{attribute 'GeneratedUsingTerminal: EK1100-0000-0018'}
{attribute addProperty BoxType "EK1100-0000-0018"}
{attribute addProperty Id "Term_882_EL1809EL1809_32157CFD20Term_883_EL1809EL1809_32157CFD20Term_884_EL1809EL1809_32157CFD20Term_885_EL1809EL1809_32157CFD20Term_886_EL1809EL1809_32157CFD20Term_887_EL1809EL1809_32157CFD20Term_888_EL1809EL1809_32157CFD20Term_889_EL1809EL1809_32157CFD20Term_890_EL1809EL1809_32157CFD20Term_891_EL1809EL1809_32157CFD20Term_892_EL1809EL1809_32157CFD20Term_893_EL1809EL1809_32157CFD20Term_894_EL1809EL1809_32157CFD20Term_895_EL1809EL1809_32157CFD20Term_896_EL1809EL1809_32157CFD20Term_897_EL1809EL1809_32157CFD20Term_898_EL1809EL1809_32157CFD20Term_899_EL1809EL1809_32157CFD20Term_900_EL1809EL1809_32157CFD20Term_901_EL1809EL1809_32157CFD20Term_902_EL1809EL1809_32157CFD20Term_903_EL1809EL1809_32157CFD20Term_904_EL1809EL1809_32157CFD20Term_905_EL1809EL1809_32157CFD20Term_906_EL1809EL1809_32157CFD20Term_933_EL1809EL1809_32157CFD20Term_934_EL1809EL1809_32157CFD20Term_935_EL1809EL1809_32157CFD20Term_936_EL1809EL1809_32157CFD20Term_937_EL1809EL1809_32157CFD20Term_938_EL1809EL1809_32157CFD20Term_939_EL1809EL1809_32157CFD20Term_940_EL1809EL1809_32157CFD20Term_941_EL1809EL1809_32157CFD20Term_942_EL1809EL1809_32157CFD20Term_943_EL1809EL1809_32157CFD20Term_944_EL1809EL1809_32157CFD20Term_945_EL1809EL1809_32157CFD20Term_946_EL1809EL1809_32157CFD20Term_947_EL1809EL1809_32157CFD20Term_948_EL1809EL1809_32157CFD20Term_949_EL1809EL1809_32157CFD20Term_950_EL1809EL1809_32157CFD20Term_951_EL1809EL1809_32157CFD20Term_952_EL1809EL1809_32157CFD20Term_953_EL1809EL1809_32157CFD20Term_954_EL1809EL1809_32157CFD20Term_955_EL1809EL1809_32157CFD20Term_956_EL1809EL1809_32157CFD20Term_957_EL1809EL1809_32157CFD20Term_958_EL1809EL1809_32157CFD20Term_959_EL1809EL1809_32157CFD20Term_960_EL1809EL1809_32157CFD20Term_961_EL1809EL1809_32157CFD20Term_962_EL1809EL1809_32157CFD20Term_963_EL1809EL1809_32157CFD20Term_964_EL1809EL1809_32157CFD20Term_965_EL1809EL1809_32157CFD20Term_967_EL1809EL1809_32157CFD20Term_968_EL1809EL1809_32157CFD20Term_969_EL1809EL1809_32157CFD20Term_970_EL1809EL1809_32157CFD20Term_971_EL1809EL1809_32157CFD20Term_972_EL1809EL1809_32157CFD20Term_973_EL1809EL1809_32157CFD20Term_974_EL1809EL1809_32157CFD20Term_975_EL1809EL1809_32157CFD20Term_976_EL1809EL1809_32157CFD20Term_977_EL1809EL1809_32157CFD20Term_978_EL1809EL1809_32157CFD20Term_979_EL1809EL1809_32157CFD20Term_980_EL1809EL1809_32157CFD20Term_981_EL1809EL1809_32157CFD20Term_982_EL1809EL1809_32157CFD20Term_983_EL1809EL1809_32157CFD20Term_984_EL1809EL1809_32157CFD20Term_986_EL1809EL1809_32157CFD20Term_987_EL1809EL1809_32157CFD20Term_988_EL1809EL1809_32157CFD20Term_989_EL1809EL1809_32157CFD20Term_1025_EL1809EL1809_32157CFD20Term_1026_EL1809EL1809_32157CFD20Term_1027_EL1809EL1809_32157CFD20Term_1028_EL1809EL1809_32157CFD20Term_1029_EL1809EL1809_32157CFD20Term_1030_EL1809EL1809_32157CFD20Term_1031_EL1809EL1809_32157CFD20Term_1032_EL1809EL1809_32157CFD20Term_1033_EL1809EL1809_32157CFD20Term_1034_EL1809EL1809_32157CFD20Term_1035_EL1809EL1809_32157CFD20Term_1036_EL1809EL1809_32157CFD20Term_1038_EL1809EL1809_32157CFD20Term_1039_EL1809EL1809_32157CFD20Term_1040_EL1809EL1809_32157CFD20Term_1041_EL1809EL1809_32157CFD20Term_1042_EL1809EL1809_32157CFD20Term_1043_EL1809EL1809_32157CFD20Term_1044_EL1809EL1809_32157CFD20Term_1045_EL1809EL1809_32157CFD20Term_1046_EK1110EK1110_1FC0878B2"}
{attribute addProperty CRC "4147311472"}
{attribute addProperty Size "2002"}
{attribute addProperty Name "Term 881 (EK1100)"}
TYPE Term_881_EK1100_F732F370 EXTENDS EK1100_1FC0878B :
STRUCT
	{attribute addProperty Name "Term 882 (EL1809)"}
	{attribute addProperty PreviousPort "Term 881 (EK1100) : B"}
	{attribute addProperty SyncUnit "default"}
	Term_882_EL1809 : EL1809_32157CFD;
	{attribute addProperty Name "Term 883 (EL1809)"}
	{attribute addProperty PreviousPort "Term 882 (EL1809) : B"}
	{attribute addProperty SyncUnit "default"}
	Term_883_EL1809 : EL1809_32157CFD;
	{attribute addProperty Name "Term 884 (EL1809)"}
	{attribute addProperty PreviousPort "Term 883 (EL1809) : B"}
	{attribute addProperty SyncUnit "default"}
	Term_884_EL1809 : EL1809_32157CFD;
	{attribute addProperty Name "Term 885 (EL1809)"}
	{attribute addProperty PreviousPort "Term 884 (EL1809) : B"}
	{attribute addProperty SyncUnit "default"}
	Term_885_EL1809 : EL1809_32157CFD;
	{attribute addProperty Name "Term 886 (EL1809)"}
	{attribute addProperty PreviousPort "Term 885 (EL1809) : B"}
	{attribute addProperty SyncUnit "default"}
	Term_886_EL1809 : EL1809_32157CFD;
	{attribute addProperty Name "Term 887 (EL1809)"}
	{attribute addProperty PreviousPort "Term 886 (EL1809) : B"}
	{attribute addProperty SyncUnit "default"}
	Term_887_EL1809 : EL1809_32157CFD;
	{attribute addProperty Name "Term 888 (EL1809)"}
	{attribute addProperty PreviousPort "Term 887 (EL1809) : B"}
	{attribute addProperty SyncUnit "default"}
	Term_888_EL1809 : EL1809_32157CFD;
	{attribute addProperty Name "Term 889 (EL1809)"}
	{attribute addProperty PreviousPort "Term 888 (EL1809) : B"}
	{attribute addProperty SyncUnit "default"}
	Term_889_EL1809 : EL1809_32157CFD;
	{attribute addProperty Name "Term 890 (EL1809)"}
	{attribute addProperty PreviousPort "Term 889 (EL1809) : B"}
	{attribute addProperty SyncUnit "default"}
	Term_890_EL1809 : EL1809_32157CFD;
	{attribute addProperty Name "Term 891 (EL1809)"}
	{attribute addProperty PreviousPort "Term 890 (EL1809) : B"}
	{attribute addProperty SyncUnit "default"}
	Term_891_EL1809 : EL1809_32157CFD;
	{attribute addProperty Name "Term 892 (EL1809)"}
	{attribute addProperty PreviousPort "Term 891 (EL1809) : B"}
	{attribute addProperty SyncUnit "default"}
	Term_892_EL1809 : EL1809_32157CFD;
	{attribute addProperty Name "Term 893 (EL1809)"}
	{attribute addProperty PreviousPort "Term 892 (EL1809) : B"}
	{attribute addProperty SyncUnit "default"}
	Term_893_EL1809 : EL1809_32157CFD;
	{attribute addProperty Name "Term 894 (EL1809)"}
	{attribute addProperty PreviousPort "Term 893 (EL1809) : B"}
	{attribute addProperty SyncUnit "default"}
	Term_894_EL1809 : EL1809_32157CFD;
	{attribute addProperty Name "Term 895 (EL1809)"}
	{attribute addProperty PreviousPort "Term 894 (EL1809) : B"}
	{attribute addProperty SyncUnit "default"}
	Term_895_EL1809 : EL1809_32157CFD;
	{attribute addProperty Name "Term 896 (EL1809)"}
	{attribute addProperty PreviousPort "Term 895 (EL1809) : B"}
	{attribute addProperty SyncUnit "default"}
	Term_896_EL1809 : EL1809_32157CFD;
	{attribute addProperty Name "Term 897 (EL1809)"}
	{attribute addProperty PreviousPort "Term 896 (EL1809) : B"}
	{attribute addProperty SyncUnit "default"}
	Term_897_EL1809 : EL1809_32157CFD;
	{attribute addProperty Name "Term 898 (EL1809)"}
	{attribute addProperty PreviousPort "Term 897 (EL1809) : B"}
	{attribute addProperty SyncUnit "default"}
	Term_898_EL1809 : EL1809_32157CFD;
	{attribute addProperty Name "Term 899 (EL1809)"}
	{attribute addProperty PreviousPort "Term 898 (EL1809) : B"}
	{attribute addProperty SyncUnit "default"}
	Term_899_EL1809 : EL1809_32157CFD;
	{attribute addProperty Name "Term 900 (EL1809)"}
	{attribute addProperty PreviousPort "Term 899 (EL1809) : B"}
	{attribute addProperty SyncUnit "default"}
	Term_900_EL1809 : EL1809_32157CFD;
	{attribute addProperty Name "Term 901 (EL1809)"}
	{attribute addProperty PreviousPort "Term 900 (EL1809) : B"}
	{attribute addProperty SyncUnit "default"}
	Term_901_EL1809 : EL1809_32157CFD;
	{attribute addProperty Name "Term 902 (EL1809)"}
	{attribute addProperty PreviousPort "Term 901 (EL1809) : B"}
	{attribute addProperty SyncUnit "default"}
	Term_902_EL1809 : EL1809_32157CFD;
	{attribute addProperty Name "Term 903 (EL1809)"}
	{attribute addProperty PreviousPort "Term 902 (EL1809) : B"}
	{attribute addProperty SyncUnit "default"}
	Term_903_EL1809 : EL1809_32157CFD;
	{attribute addProperty Name "Term 904 (EL1809)"}
	{attribute addProperty PreviousPort "Term 903 (EL1809) : B"}
	{attribute addProperty SyncUnit "default"}
	Term_904_EL1809 : EL1809_32157CFD;
	{attribute addProperty Name "Term 905 (EL1809)"}
	{attribute addProperty PreviousPort "Term 904 (EL1809) : B"}
	{attribute addProperty SyncUnit "default"}
	Term_905_EL1809 : EL1809_32157CFD;
	{attribute addProperty Name "Term 906 (EL1809)"}
	{attribute addProperty PreviousPort "Term 905 (EL1809) : B"}
	{attribute addProperty SyncUnit "default"}
	Term_906_EL1809 : EL1809_32157CFD;
	{attribute addProperty Name "Term 933 (EL1809)"}
	{attribute addProperty PreviousPort "Term 906 (EL1809) : B"}
	{attribute addProperty SyncUnit "default"}
	Term_933_EL1809 : EL1809_32157CFD;
	{attribute addProperty Name "Term 934 (EL1809)"}
	{attribute addProperty PreviousPort "Term 933 (EL1809) : B"}
	{attribute addProperty SyncUnit "default"}
	Term_934_EL1809 : EL1809_32157CFD;
	{attribute addProperty Name "Term 935 (EL1809)"}
	{attribute addProperty PreviousPort "Term 934 (EL1809) : B"}
	{attribute addProperty SyncUnit "default"}
	Term_935_EL1809 : EL1809_32157CFD;
	{attribute addProperty Name "Term 936 (EL1809)"}
	{attribute addProperty PreviousPort "Term 935 (EL1809) : B"}
	{attribute addProperty SyncUnit "default"}
	Term_936_EL1809 : EL1809_32157CFD;
	{attribute addProperty Name "Term 937 (EL1809)"}
	{attribute addProperty PreviousPort "Term 936 (EL1809) : B"}
	{attribute addProperty SyncUnit "default"}
	Term_937_EL1809 : EL1809_32157CFD;
	{attribute addProperty Name "Term 938 (EL1809)"}
	{attribute addProperty PreviousPort "Term 937 (EL1809) : B"}
	{attribute addProperty SyncUnit "default"}
	Term_938_EL1809 : EL1809_32157CFD;
	{attribute addProperty Name "Term 939 (EL1809)"}
	{attribute addProperty PreviousPort "Term 938 (EL1809) : B"}
	{attribute addProperty SyncUnit "default"}
	Term_939_EL1809 : EL1809_32157CFD;
	{attribute addProperty Name "Term 940 (EL1809)"}
	{attribute addProperty PreviousPort "Term 939 (EL1809) : B"}
	{attribute addProperty SyncUnit "default"}
	Term_940_EL1809 : EL1809_32157CFD;
	{attribute addProperty Name "Term 941 (EL1809)"}
	{attribute addProperty PreviousPort "Term 940 (EL1809) : B"}
	{attribute addProperty SyncUnit "default"}
	Term_941_EL1809 : EL1809_32157CFD;
	{attribute addProperty Name "Term 942 (EL1809)"}
	{attribute addProperty PreviousPort "Term 941 (EL1809) : B"}
	{attribute addProperty SyncUnit "default"}
	Term_942_EL1809 : EL1809_32157CFD;
	{attribute addProperty Name "Term 943 (EL1809)"}
	{attribute addProperty PreviousPort "Term 942 (EL1809) : B"}
	{attribute addProperty SyncUnit "default"}
	Term_943_EL1809 : EL1809_32157CFD;
	{attribute addProperty Name "Term 944 (EL1809)"}
	{attribute addProperty PreviousPort "Term 943 (EL1809) : B"}
	{attribute addProperty SyncUnit "default"}
	Term_944_EL1809 : EL1809_32157CFD;
	{attribute addProperty Name "Term 945 (EL1809)"}
	{attribute addProperty PreviousPort "Term 944 (EL1809) : B"}
	{attribute addProperty SyncUnit "default"}
	Term_945_EL1809 : EL1809_32157CFD;
	{attribute addProperty Name "Term 946 (EL1809)"}
	{attribute addProperty PreviousPort "Term 945 (EL1809) : B"}
	{attribute addProperty SyncUnit "default"}
	Term_946_EL1809 : EL1809_32157CFD;
	{attribute addProperty Name "Term 947 (EL1809)"}
	{attribute addProperty PreviousPort "Term 946 (EL1809) : B"}
	{attribute addProperty SyncUnit "default"}
	Term_947_EL1809 : EL1809_32157CFD;
	{attribute addProperty Name "Term 948 (EL1809)"}
	{attribute addProperty PreviousPort "Term 947 (EL1809) : B"}
	{attribute addProperty SyncUnit "default"}
	Term_948_EL1809 : EL1809_32157CFD;
	{attribute addProperty Name "Term 949 (EL1809)"}
	{attribute addProperty PreviousPort "Term 948 (EL1809) : B"}
	{attribute addProperty SyncUnit "default"}
	Term_949_EL1809 : EL1809_32157CFD;
	{attribute addProperty Name "Term 950 (EL1809)"}
	{attribute addProperty PreviousPort "Term 949 (EL1809) : B"}
	{attribute addProperty SyncUnit "default"}
	Term_950_EL1809 : EL1809_32157CFD;
	{attribute addProperty Name "Term 951 (EL1809)"}
	{attribute addProperty PreviousPort "Term 950 (EL1809) : B"}
	{attribute addProperty SyncUnit "default"}
	Term_951_EL1809 : EL1809_32157CFD;
	{attribute addProperty Name "Term 952 (EL1809)"}
	{attribute addProperty PreviousPort "Term 951 (EL1809) : B"}
	{attribute addProperty SyncUnit "default"}
	Term_952_EL1809 : EL1809_32157CFD;
	{attribute addProperty Name "Term 953 (EL1809)"}
	{attribute addProperty PreviousPort "Term 952 (EL1809) : B"}
	{attribute addProperty SyncUnit "default"}
	Term_953_EL1809 : EL1809_32157CFD;
	{attribute addProperty Name "Term 954 (EL1809)"}
	{attribute addProperty PreviousPort "Term 953 (EL1809) : B"}
	{attribute addProperty SyncUnit "default"}
	Term_954_EL1809 : EL1809_32157CFD;
	{attribute addProperty Name "Term 955 (EL1809)"}
	{attribute addProperty PreviousPort "Term 954 (EL1809) : B"}
	{attribute addProperty SyncUnit "default"}
	Term_955_EL1809 : EL1809_32157CFD;
	{attribute addProperty Name "Term 956 (EL1809)"}
	{attribute addProperty PreviousPort "Term 955 (EL1809) : B"}
	{attribute addProperty SyncUnit "default"}
	Term_956_EL1809 : EL1809_32157CFD;
	{attribute addProperty Name "Term 957 (EL1809)"}
	{attribute addProperty PreviousPort "Term 956 (EL1809) : B"}
	{attribute addProperty SyncUnit "default"}
	Term_957_EL1809 : EL1809_32157CFD;
	{attribute addProperty Name "Term 958 (EL1809)"}
	{attribute addProperty PreviousPort "Term 957 (EL1809) : B"}
	{attribute addProperty SyncUnit "default"}
	Term_958_EL1809 : EL1809_32157CFD;
	{attribute addProperty Name "Term 959 (EL1809)"}
	{attribute addProperty PreviousPort "Term 958 (EL1809) : B"}
	{attribute addProperty SyncUnit "default"}
	Term_959_EL1809 : EL1809_32157CFD;
	{attribute addProperty Name "Term 960 (EL1809)"}
	{attribute addProperty PreviousPort "Term 959 (EL1809) : B"}
	{attribute addProperty SyncUnit "default"}
	Term_960_EL1809 : EL1809_32157CFD;
	{attribute addProperty Name "Term 961 (EL1809)"}
	{attribute addProperty PreviousPort "Term 960 (EL1809) : B"}
	{attribute addProperty SyncUnit "default"}
	Term_961_EL1809 : EL1809_32157CFD;
	{attribute addProperty Name "Term 962 (EL1809)"}
	{attribute addProperty PreviousPort "Term 961 (EL1809) : B"}
	{attribute addProperty SyncUnit "default"}
	Term_962_EL1809 : EL1809_32157CFD;
	{attribute addProperty Name "Term 963 (EL1809)"}
	{attribute addProperty PreviousPort "Term 962 (EL1809) : B"}
	{attribute addProperty SyncUnit "default"}
	Term_963_EL1809 : EL1809_32157CFD;
	{attribute addProperty Name "Term 964 (EL1809)"}
	{attribute addProperty PreviousPort "Term 963 (EL1809) : B"}
	{attribute addProperty SyncUnit "default"}
	Term_964_EL1809 : EL1809_32157CFD;
	{attribute addProperty Name "Term 965 (EL1809)"}
	{attribute addProperty PreviousPort "Term 964 (EL1809) : B"}
	{attribute addProperty SyncUnit "default"}
	Term_965_EL1809 : EL1809_32157CFD;
	{attribute addProperty Name "Term 967 (EL1809)"}
	{attribute addProperty PreviousPort "Term 965 (EL1809) : B"}
	{attribute addProperty SyncUnit "default"}
	Term_967_EL1809 : EL1809_32157CFD;
	{attribute addProperty Name "Term 968 (EL1809)"}
	{attribute addProperty PreviousPort "Term 967 (EL1809) : B"}
	{attribute addProperty SyncUnit "default"}
	Term_968_EL1809 : EL1809_32157CFD;
	{attribute addProperty Name "Term 969 (EL1809)"}
	{attribute addProperty PreviousPort "Term 968 (EL1809) : B"}
	{attribute addProperty SyncUnit "default"}
	Term_969_EL1809 : EL1809_32157CFD;
	{attribute addProperty Name "Term 970 (EL1809)"}
	{attribute addProperty PreviousPort "Term 969 (EL1809) : B"}
	{attribute addProperty SyncUnit "default"}
	Term_970_EL1809 : EL1809_32157CFD;
	{attribute addProperty Name "Term 971 (EL1809)"}
	{attribute addProperty PreviousPort "Term 970 (EL1809) : B"}
	{attribute addProperty SyncUnit "default"}
	Term_971_EL1809 : EL1809_32157CFD;
	{attribute addProperty Name "Term 972 (EL1809)"}
	{attribute addProperty PreviousPort "Term 971 (EL1809) : B"}
	{attribute addProperty SyncUnit "default"}
	Term_972_EL1809 : EL1809_32157CFD;
	{attribute addProperty Name "Term 973 (EL1809)"}
	{attribute addProperty PreviousPort "Term 972 (EL1809) : B"}
	{attribute addProperty SyncUnit "default"}
	Term_973_EL1809 : EL1809_32157CFD;
	{attribute addProperty Name "Term 974 (EL1809)"}
	{attribute addProperty PreviousPort "Term 973 (EL1809) : B"}
	{attribute addProperty SyncUnit "default"}
	Term_974_EL1809 : EL1809_32157CFD;
	{attribute addProperty Name "Term 975 (EL1809)"}
	{attribute addProperty PreviousPort "Term 974 (EL1809) : B"}
	{attribute addProperty SyncUnit "default"}
	Term_975_EL1809 : EL1809_32157CFD;
	{attribute addProperty Name "Term 976 (EL1809)"}
	{attribute addProperty PreviousPort "Term 975 (EL1809) : B"}
	{attribute addProperty SyncUnit "default"}
	Term_976_EL1809 : EL1809_32157CFD;
	{attribute addProperty Name "Term 977 (EL1809)"}
	{attribute addProperty PreviousPort "Term 976 (EL1809) : B"}
	{attribute addProperty SyncUnit "default"}
	Term_977_EL1809 : EL1809_32157CFD;
	{attribute addProperty Name "Term 978 (EL1809)"}
	{attribute addProperty PreviousPort "Term 977 (EL1809) : B"}
	{attribute addProperty SyncUnit "default"}
	Term_978_EL1809 : EL1809_32157CFD;
	{attribute addProperty Name "Term 979 (EL1809)"}
	{attribute addProperty PreviousPort "Term 978 (EL1809) : B"}
	{attribute addProperty SyncUnit "default"}
	Term_979_EL1809 : EL1809_32157CFD;
	{attribute addProperty Name "Term 980 (EL1809)"}
	{attribute addProperty PreviousPort "Term 979 (EL1809) : B"}
	{attribute addProperty SyncUnit "default"}
	Term_980_EL1809 : EL1809_32157CFD;
	{attribute addProperty Name "Term 981 (EL1809)"}
	{attribute addProperty PreviousPort "Term 980 (EL1809) : B"}
	{attribute addProperty SyncUnit "default"}
	Term_981_EL1809 : EL1809_32157CFD;
	{attribute addProperty Name "Term 982 (EL1809)"}
	{attribute addProperty PreviousPort "Term 981 (EL1809) : B"}
	{attribute addProperty SyncUnit "default"}
	Term_982_EL1809 : EL1809_32157CFD;
	{attribute addProperty Name "Term 983 (EL1809)"}
	{attribute addProperty PreviousPort "Term 982 (EL1809) : B"}
	{attribute addProperty SyncUnit "default"}
	Term_983_EL1809 : EL1809_32157CFD;
	{attribute addProperty Name "Term 984 (EL1809)"}
	{attribute addProperty PreviousPort "Term 983 (EL1809) : B"}
	{attribute addProperty SyncUnit "default"}
	Term_984_EL1809 : EL1809_32157CFD;
	{attribute addProperty Name "Term 986 (EL1809)"}
	{attribute addProperty PreviousPort "Term 984 (EL1809) : B"}
	{attribute addProperty SyncUnit "default"}
	Term_986_EL1809 : EL1809_32157CFD;
	{attribute addProperty Name "Term 987 (EL1809)"}
	{attribute addProperty PreviousPort "Term 986 (EL1809) : B"}
	{attribute addProperty SyncUnit "default"}
	Term_987_EL1809 : EL1809_32157CFD;
	{attribute addProperty Name "Term 988 (EL1809)"}
	{attribute addProperty PreviousPort "Term 987 (EL1809) : B"}
	{attribute addProperty SyncUnit "default"}
	Term_988_EL1809 : EL1809_32157CFD;
	{attribute addProperty Name "Term 989 (EL1809)"}
	{attribute addProperty PreviousPort "Term 988 (EL1809) : B"}
	{attribute addProperty SyncUnit "default"}
	Term_989_EL1809 : EL1809_32157CFD;
	{attribute addProperty Name "Term 1025 (EL1809)"}
	{attribute addProperty PreviousPort "Term 989 (EL1809) : B"}
	{attribute addProperty SyncUnit "default"}
	Term_1025_EL1809 : EL1809_32157CFD;
	{attribute addProperty Name "Term 1026 (EL1809)"}
	{attribute addProperty PreviousPort "Term 1025 (EL1809) : B"}
	{attribute addProperty SyncUnit "default"}
	Term_1026_EL1809 : EL1809_32157CFD;
	{attribute addProperty Name "Term 1027 (EL1809)"}
	{attribute addProperty PreviousPort "Term 1026 (EL1809) : B"}
	{attribute addProperty SyncUnit "default"}
	Term_1027_EL1809 : EL1809_32157CFD;
	{attribute addProperty Name "Term 1028 (EL1809)"}
	{attribute addProperty PreviousPort "Term 1027 (EL1809) : B"}
	{attribute addProperty SyncUnit "default"}
	Term_1028_EL1809 : EL1809_32157CFD;
	{attribute addProperty Name "Term 1029 (EL1809)"}
	{attribute addProperty PreviousPort "Term 1028 (EL1809) : B"}
	{attribute addProperty SyncUnit "default"}
	Term_1029_EL1809 : EL1809_32157CFD;
	{attribute addProperty Name "Term 1030 (EL1809)"}
	{attribute addProperty PreviousPort "Term 1029 (EL1809) : B"}
	{attribute addProperty SyncUnit "default"}
	Term_1030_EL1809 : EL1809_32157CFD;
	{attribute addProperty Name "Term 1031 (EL1809)"}
	{attribute addProperty PreviousPort "Term 1030 (EL1809) : B"}
	{attribute addProperty SyncUnit "default"}
	Term_1031_EL1809 : EL1809_32157CFD;
	{attribute addProperty Name "Term 1032 (EL1809)"}
	{attribute addProperty PreviousPort "Term 1031 (EL1809) : B"}
	{attribute addProperty SyncUnit "default"}
	Term_1032_EL1809 : EL1809_32157CFD;
	{attribute addProperty Name "Term 1033 (EL1809)"}
	{attribute addProperty PreviousPort "Term 1032 (EL1809) : B"}
	{attribute addProperty SyncUnit "default"}
	Term_1033_EL1809 : EL1809_32157CFD;
	{attribute addProperty Name "Term 1034 (EL1809)"}
	{attribute addProperty PreviousPort "Term 1033 (EL1809) : B"}
	{attribute addProperty SyncUnit "default"}
	Term_1034_EL1809 : EL1809_32157CFD;
	{attribute addProperty Name "Term 1035 (EL1809)"}
	{attribute addProperty PreviousPort "Term 1034 (EL1809) : B"}
	{attribute addProperty SyncUnit "default"}
	Term_1035_EL1809 : EL1809_32157CFD;
	{attribute addProperty Name "Term 1036 (EL1809)"}
	{attribute addProperty PreviousPort "Term 1035 (EL1809) : B"}
	{attribute addProperty SyncUnit "default"}
	Term_1036_EL1809 : EL1809_32157CFD;
	{attribute addProperty Name "Term 1038 (EL1809)"}
	{attribute addProperty PreviousPort "Term 1036 (EL1809) : B"}
	{attribute addProperty SyncUnit "default"}
	Term_1038_EL1809 : EL1809_32157CFD;
	{attribute addProperty Name "Term 1039 (EL1809)"}
	{attribute addProperty PreviousPort "Term 1038 (EL1809) : B"}
	{attribute addProperty SyncUnit "default"}
	Term_1039_EL1809 : EL1809_32157CFD;
	{attribute addProperty Name "Term 1040 (EL1809)"}
	{attribute addProperty PreviousPort "Term 1039 (EL1809) : B"}
	{attribute addProperty SyncUnit "default"}
	Term_1040_EL1809 : EL1809_32157CFD;
	{attribute addProperty Name "Term 1041 (EL1809)"}
	{attribute addProperty PreviousPort "Term 1040 (EL1809) : B"}
	{attribute addProperty SyncUnit "default"}
	Term_1041_EL1809 : EL1809_32157CFD;
	{attribute addProperty Name "Term 1042 (EL1809)"}
	{attribute addProperty PreviousPort "Term 1041 (EL1809) : B"}
	{attribute addProperty SyncUnit "default"}
	Term_1042_EL1809 : EL1809_32157CFD;
	{attribute addProperty Name "Term 1043 (EL1809)"}
	{attribute addProperty PreviousPort "Term 1042 (EL1809) : B"}
	{attribute addProperty SyncUnit "default"}
	Term_1043_EL1809 : EL1809_32157CFD;
	{attribute addProperty Name "Term 1044 (EL1809)"}
	{attribute addProperty PreviousPort "Term 1043 (EL1809) : B"}
	{attribute addProperty SyncUnit "default"}
	Term_1044_EL1809 : EL1809_32157CFD;
	{attribute addProperty Name "Term 1045 (EL1809)"}
	{attribute addProperty PreviousPort "Term 1044 (EL1809) : B"}
	{attribute addProperty SyncUnit "default"}
	Term_1045_EL1809 : EL1809_32157CFD;
	{attribute addProperty Name "Term 1046 (EK1110)"}
	{attribute addProperty PreviousPort "Term 1045 (EL1809) : B"}
	{attribute addProperty SyncUnit "default"}
	Term_1046_EK1110 : EK1110_1FC0878B;
END_STRUCT
END_TYPE

(* stored: Version 1.2.0.0, ProductVersion 3.1.4024.11
   DUT Term_881_EK1100_F732F370: Id {ea615791-79e2-0625-064b-c340df52f82e} *)
